{attribute 'no_check'}
FUNCTION_BLOCK EcSlaveInfoData implements I_EcSlaveInfoData
VAR_INPUT
END_VAR
VAR_OUTPUT
	WcState											AT  %I*		:	BOOL;			//TRUE=Invalid - TRUE an invalid working counter and FALSE a valid working counter 
	InputToggle										AT  %I*		:	BOOL;			//variable toggles in every successful cycle	
	{attribute 'displaymode':='hex'}  
	InfoDataState									AT  %I*		: 	UINT;			(* current EtherCAT device state:
																						EC_DEVICE_STATE_MASK		:BYTE 	:=16#0F;
																						EC_DEVICE_STATE_INIT		:BYTE 	:=16#01;
																						EC_DEVICE_STATE_PREOP		:BYTE 	:=16#02;
																						EC_DEVICE_STATE_BOOTSTRAP	:BYTE 	:=16#03;
																						EC_DEVICE_STATE_SAFEOP		:BYTE 	:=16#04;
																						EC_DEVICE_STATE_OP			:BYTE 	:=16#08;
																						EC_DEVICE_STATE_ERROR		:BYTE 	:=16#10;
																						EC_DEVICE_STATE_INVALID_VPRS :BYTE 	:=16#20;
																						EC_DEVICE_STATE_INITCMD_ERROR:BYTE 	:=16#40; *)
	AdsAddr											AT  %I*		:	AMSADDR; 		//Slave device AdsAddr structure(ID and port number)
END_VAR
VAR
END_VAR

;

PROPERTY PUBLIC rInfoData : reference to EcSlaveInfoData
GET
rInfoData := THis^;
END_GET
END_PROPERTY

END_FUNCTION_BLOCK

(* stored: Version 1.1.0.1, ProductVersion 3.1.4024.6
   POU EcSlaveInfoData: Id {abde7282-e04f-42c5-8dbe-db29c91a0248}, SpecialFunc None
   Property rInfoData: Id {e69e7ae9-95ed-4260-8d4f-aebfc81bd379}
   Get Get: Id {9c1529c7-eb6f-47ad-87a2-7e3936964c78} *)
